FUNCTION_BLOCK FB_WorkerDefGrid_Delete EXTENDS FB_WorkerDefGrid
VAR PERSISTENT
  _fWorkerToPu   : LREAL := 3;    (*Distance between PU and this worker, mechanisch*)
END_VAR

METHOD PROTECTED  Attach : BOOL
VAR_INPUT
  iCT              : I_CT;                         (*container at triggered event position*)
END_VAR
IF SUPER^.Attach(iCT:=iCT) THEN
  ;
END_IF
END_METHOD

PROPERTY fWorkerToPu : LREAL
GET
fWorkerToPu := _fWorkerToPu;
END_GET
END_PROPERTY

METHOD   mJobStart
VAR_INPUT
	sJobDef	: CalmarCompPrint.I_JobDefinition;
END_VAR

_bJobActive := TRUE;
END_METHOD

METHOD  mJobStop
VAR_INPUT
	sStatus	: CalmarCompPrint.I_JobStatus;
END_VAR
_bJobActive := FALSE;
END_METHOD

METHOD Release : BOOL
VAR_INPUT
  iCT              : I_CT;                         (*container at triggered event position*)
END_VAR
IF SUPER^.Release(iCT := iCT) THEN
  
  // it's the last worker so distroy attached CT
  IF _pCtManager <> 0 THEN
    LogLvl(Lvl:=E_LogSeverity.Debug, Msg:=F_Concat2('DestroyCT: ', TO_STRING(iCT.pCT^.iId)));
    _pCtManager^.DestroyCT(iCT:=iCT);
  END_IF
  
END_IF
END_METHOD

METHOD  work
SUPER^.work();

//Worker position update
IF _pParamMediator <> 0 AND _pAttachedCt = 0 THEN     // Update only without attached container
  // WorkerPosition =  Worker<-PU<-CAM<-SheetDetect
  fPosition := _fWorkerToPu + _pParamMediator^.fCameraToPrintOffset + _pParamMediator^.fDetectToCamera;
END_IF

IF _pAttachedCt <> 0 THEN
  Release(iCT:=_pAttachedCt^);
END_IF
END_METHOD

END_FUNCTION_BLOCK

(* stored: Version 1.1.0.1, ProductVersion 3.1.4024.3
   POU FB_WorkerDefGrid_Delete: Id {7527e8ae-b298-40c4-9d5c-225c5c9f33be}, SpecialFunc None
   Method Attach: Id {ba44b2bb-b602-4351-b884-27d38546747f}
   Property fWorkerToPu: Id {89984a29-c49f-4fef-962c-903196b3c502}
   Get Get: Id {69475d99-e2f1-4a28-885b-7624fa90c9a3}
   Method mJobStart: Id {35dee294-0abe-481b-9d05-6c256fb62d03}
   Method mJobStop: Id {78e31b74-c4ab-4dcf-9c3a-eb2545757f78}
   Method Release: Id {7ef7389d-1596-4a7c-82f8-404606f272e5}
   Method work: Id {7026ea79-caca-4595-a7ed-707178d44865} *)
